FUNCTION_BLOCK F_BOOL_AS_STRING (* Convert BOOL to STRING *)
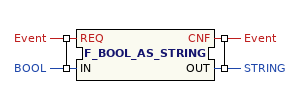
  EVENT_INPUT
    REQ WITH IN; (* Normal Execution Request *)
  END_EVENT
  EVENT_OUTPUT
    CNF WITH OUT; (* Execution Confirmation *)
  END_EVENT
  VAR_INPUT
    IN : BOOL;
  END_VAR
  VAR_OUTPUT
    OUT : STRING;
  END_VAR
  ALGORITHM REQ IN ST:
OUT := BOOL_AS_STRING(IN);
  END_ALGORITHM
END_FUNCTION_BLOCK
